# EPICS autosave request: ads-ioc/valveApp/Db/valve.req
$(P):CycleCounter.VAL
$(P):OpenTimeTotal.VAL
